// TIA Portal V19 export
DATA_BLOCK "F_DB"   // DB2, F_DB
// stored: Access Published
   VAR
      SafetyReset : Bool;   // Cumulative safety reset
      SuperUserReset : Bool;   // Cumulative super user safety reset
      Enable_Reset_Superuser : Bool := TRUE;
      A01_Estop : Bool;   // Emergency stop to Area 01 (1=No stop)
      A01_EstopDelay : Bool;   // Emergency stop delayed to Area 01 (1=No stop)
      A02_Estop : Bool;   // Emergency stop to Area 02 (1=No stop)
      A02_EstopDelay : Bool;   // Emergency stop delayed to Area 02 (1=No stop)
      A03_Estop : Bool;   // Emergency stop to Area 03 (1=No stop)
      A03_EstopDelay : Bool;   // Emergency stop delayed to Area 03 (1=No stop)
      LB101 : "udt_BimanualSts";   // LB101 Two hands @ Zone 01 (Front of decoiler in load)
      LB111 : "udt_BimanualSts";   // LB111 Two hands @ Zone 00 (Coil Car)
      LB112 : "udt_BimanualSts";   // LB112 Two Hands @ Zone 05 FRONT (Straightner entry) used for operations inside Zone 05
      LB113 : "udt_BimanualSts";   // LB113 Two Hands @ Zone 05 FRONT (Junction bench) used for operations inside Zone 05
      LB113_W : "udt_BimanualSts";   // LB113 Enabling switch @ Zone 05 FRONT (Junction bench) used for welding operations
      LB114_FeedA01 : "udt_BimanualSts";   // LB114 Two Hands @ Zone 05 FRONT (Loop 1 / Rollformer entry) used for A01 Material feeding
      LB114_FeedA02 : "udt_BimanualSts";   // LB114 Two Hands @ Zone 05 FRONT (Loop 1 / Rollformer entry) used for A02 Material feeding
      LB131 : "udt_BimanualSts";   // LB131 Two Hands @ Zone 05 REAR (piantana) used for operations inside Zone 05
      LB211 : "udt_BimanualSts";   // LB211 Dead man @ Area 02 Zone xx (Rollformer)
      LB212 : "udt_BimanualSts";   // @ Hydraulic presses front (2Hands) -> Press 1 operations
      LB212_FeedA02 : "udt_BimanualSts";   // @ Hydraulic presses front (2Hands) -> Area 03 Material feeding
      LB311 : "udt_BimanualSts";   // LB311 Dead man @ Area 03 Zone xx (Bordatrice)
      D01 : "udt_DoorSts";   // A01 Light curtain (coil load side) - Ferma solo la rotazione orizzonatale / Zone 01 rear (coil handling)
      D02 : "udt_DoorSts";   // A01 Decoiler 1 in line / Zone 01 front (coil handling)
      D03 : "udt_DoorSts";   // A01 Decoiler 2 in line / Zone 02 rear (Press)
      D04 : "udt_DoorSts";   // A01 Front (Between Peeler to JB) / Zone 02 front (Press)
      D05 : "udt_DoorSts";   // A01 Rear (Between Decoiler in line to JB) / Zone 03 rear (loop 02)
      D07 : "udt_DoorSts";   // A0/A02 Rear (Loop 1)
      D10 : "udt_DoorSts";   // A02 - Front Rollformer (Entry side)
      D11 : "udt_DoorSts";   // A02 - Rear Rollformer (Exit side)
      D12 : "udt_DoorSts";   // A02 - Front Rollformer (Exit side)
      D14 : "udt_DoorSts";   // A02 - Front Flying Cut
      D15 : "udt_DoorSts";   // A02 - Rear Flying Cut
      D16 : "udt_DoorSts";   // A03 - Frinte accesso Ingresso Rulliera di accelerazione
      D18 : "udt_DoorSts";   // A03 - Fotoelettrica fronte scarico SemiGusci
      D19 : "udt_DoorSts";   // A03 - Retro accesso spintore stazione 2
      D20 : "udt_DoorSts";   // A03 - Fronte accesso Uscita Rulliera di acceleazione
      D21 : "udt_DoorSts";   // A03 - Retro accesso Bordatrice
      D22 : "udt_DoorSts";   // A03 - Accesso baia uscita esterna
      D24 : "udt_DoorSts";   // A03 - Accesso baia uscita interna
      D25 : "udt_DoorSts";   // A03 - Retri accesso accumulo Pezzi da controllare
      D27 : "udt_DoorSts";   // A03 - Testa accesso Pareggiatore / Spalle impilatore
      D30 : "udt_DoorSts";   // A02 - FAK door
      ZSI_Zone00 : "udt_ZoneSafetyInterface";   // Coil handling / A01 - Coil Car
      ZSI_Zone01 : "udt_ZoneSafetyInterface";   // Coil handling / A01 - Decoilers horizontal rotation
      ZSI_Zone02 : "udt_ZoneSafetyInterface";   // Coil handling / A01 - Decoiler 1
      ZSI_Zone03 : "udt_ZoneSafetyInterface";   // Pre-Punching press / A01 - Decoiler 2
      ZSI_Zone05 : "udt_ZoneSafetyInterface";   // Rollformer / A01 - Peelers + Straightener + JB
      ZSI_Zone06 : "udt_ZoneSafetyInterface";   // Rollformer / A01 - Loop 1
      ZSI_Zone10 : "udt_ZoneSafetyInterface";   // A01 - Material feeding & common devices
      ZSI_Zone11 : "udt_ZoneSafetyInterface";   // A02 - Rollformer
      ZSI_Zone13 : "udt_ZoneSafetyInterface";   // A02 - FlyingCut
      ZSI_Zone15 : "udt_ZoneSafetyInterface";   // A02 - Acc Rollway
      ZSI_Zone20 : "udt_ZoneSafetyInterface";   // A02 - Material feeing & common devices
      ZSI_Zone21 : "udt_ZoneSafetyInterface";   // A03 - Accoppiamento
      ZSI_Zone23 : "udt_ZoneSafetyInterface";   // A03 - Bordatrice
      ZSI_Zone25 : "udt_ZoneSafetyInterface";   // A03 - Pareggiamento
      ZSI_Zone27 : "udt_ZoneSafetyInterface";   // A03 - Creazione Pacco
      ZSI_Zone29 : "udt_ZoneSafetyInterface";   // A03 - Navetta
      FNS_Zone05 : Bool;
      FNS_Zone10 : Bool;
      FNS_Zone11 : Bool;
      FNS_Zone13 : Bool;
      FNS_Zone15 : Bool;
      FNS_Zone20 : Bool;
      FNS_Zone21 : Bool;
      FNS_Zone23 : Bool;
      FNS_Zone25 : Bool;
      FNS_Zone27 : Bool;
      FNS_Zone29 : Bool;
      DSI_V_Air_Gen : "udt_DeviceSafetyInterface";   // 0Do0
      DSI_S120_CoilCar : "udt_DeviceSafetyInterface";
      DSI_V_CoilCar : "udt_DeviceSafetyInterface";
      DSI_HU_Decoilers_Pump : "udt_DeviceSafetyInterface";   // 0Do2
      DSI_S120_Decoiler1 : "udt_DeviceSafetyInterface";
      DSI_V_Decoiler1 : "udt_DeviceSafetyInterface";   // 0Do3
      DSI_S120_Decoiler2 : "udt_DeviceSafetyInterface";
      DSI_V_Decoiler2 : "udt_DeviceSafetyInterface";   // 0Do4
      DSI_S120_DecoilersTranslation : "udt_DeviceSafetyInterface";
      DSI_V_DecoilersHorizRotation : "udt_DeviceSafetyInterface";   // 0Do1
      DSI_HU_Area01_Pump : "udt_DeviceSafetyInterface";   // 1Do3
      DSI_V_Peeler : "udt_DeviceSafetyInterface";   // 2Do2
      DSI_S120_Straightener : "udt_DeviceSafetyInterface";
      DSI_V_JB_Cut_Rest : "udt_DeviceSafetyInterface";   // 2Do0
      DSI_V_JB_Cut_Work : "udt_DeviceSafetyInterface";   // 2Do0
      DSI_S120_JB_Torch : "udt_DeviceSafetyInterface";
      DSI_S120_JB_PinchRoll : "udt_DeviceSafetyInterface";
      DSI_S120_Rollformer : "udt_DeviceSafetyInterface";
      DSI_S120_Cassetta1_OP : "udt_DeviceSafetyInterface";
      DSI_S120_Cassetta1_MOT : "udt_DeviceSafetyInterface";
      DSI_S120_Cassetta2_OP : "udt_DeviceSafetyInterface";
      DSI_S120_Cassetta2_MOT : "udt_DeviceSafetyInterface";
      DSI_S120_Cassetta3_OP : "udt_DeviceSafetyInterface";
      DSI_S120_Cassetta3_MOT : "udt_DeviceSafetyInterface";
      DSI_S120_FAK_Pusher : "udt_DeviceSafetyInterface";
      DSI_S120_Carriage : "udt_DeviceSafetyInterface";
      DSI_S120_AccRolls1 : "udt_DeviceSafetyInterface";
      DSI_S120_AccRolls2 : "udt_DeviceSafetyInterface";
      DSI_S120_AccRolls3 : "udt_DeviceSafetyInterface";
      DSI_HU_FinalCut_Pump : "udt_DeviceSafetyInterface";   // 5Do1
      DSI_V_FinalCut : "udt_DeviceSafetyInterface";
      DSI_CambioFormato_Profilatrice : "udt_DeviceSafetyInterface";   // 10Do0
      DSI_V_Air_A0301_A0302 : "udt_DeviceSafetyInterface";   // Valvola taglio aria A0301 (Ribaltamento) + A0302 ingresso (bordatrice)
      DSI_Trasporto : "udt_DeviceSafetyInterface";
      DSI_Ribaltatore : "udt_DeviceSafetyInterface";
      DSI_Spintore : "udt_DeviceSafetyInterface";
      DSI_S120_Bordatrice : "udt_DeviceSafetyInterface";
      DSI_CambioFormato_Bordatrice : "udt_DeviceSafetyInterface";   // 10Do0
      DSI_V_Air_A0302_A0303 : "udt_DeviceSafetyInterface";   // Valvola taglio aria A0302 uscita (Pareggiamemto) + A0303 (Creazione pacco)
      DSI_Rulliera1 : "udt_DeviceSafetyInterface";
      DSI_Rulliera2 : "udt_DeviceSafetyInterface";
      DSI_HU_CYTROPAC_STO : "udt_DeviceSafetyInterface";   // 5Do1
      DSI_V_PareggiatoreCoda : "udt_DeviceSafetyInterface";
      DSI_V_PareggiatoreTesta : "udt_DeviceSafetyInterface";
      DSI_PareggiatoreTesta : "udt_DeviceSafetyInterface";
      DSI_PareggiatoreCoda : "udt_DeviceSafetyInterface";
      DSI_ManipolatoreTesta : "udt_DeviceSafetyInterface";
      DSI_ManipolatoreCoda : "udt_DeviceSafetyInterface";
      DSI_SpallaTesta : "udt_DeviceSafetyInterface";
      DSI_SpallaCoda : "udt_DeviceSafetyInterface";
      DSI_TraslazioneTesta : "udt_DeviceSafetyInterface";
      DSI_TraslazioneCoda : "udt_DeviceSafetyInterface";
      DSI_SollevamentoTesta : "udt_DeviceSafetyInterface";
      DSI_SollevamentoCoda : "udt_DeviceSafetyInterface";
      DSI_SostegnoAntiribCoda : "udt_DeviceSafetyInterface";
      DSI_SostegnoAntiribTesta : "udt_DeviceSafetyInterface";
      DSI_V_Air_A0304 : "udt_DeviceSafetyInterface";
      DSI_NavettaTesta : "udt_DeviceSafetyInterface";
      DSI_NavettaCoda : "udt_DeviceSafetyInterface";
   END_VAR
BEGIN
END_DATA_BLOCK
